FUNCTION run_and_return_duration : LREAL
VAR_INPUT
  ruckig : REFERENCE TO Struckig.Ruckig;
  input : REFERENCE TO Struckig.InputParameter;
  output : REFERENCE TO Struckig.OutputParameter;  
END_VAR

WHILE(ruckig.update(input, output) = Struckig.StateEnum.busy)
DO
  input.current_position := output.new_position;
  input.current_velocity := output.new_velocity;
  input.current_acceleration := output.new_acceleration;
END_WHILE

run_and_return_duration := output.trajectory.duration;

END_FUNCTION

(* stored: Version 1.1.0.1, ProductVersion 3.1.4024.6
   POU run_and_return_duration: Id {7705c60f-b3f4-4b53-bef5-2ced749a7c74}, SpecialFunc None *)
